{attribute 'GeneratedUsingTerminal: KL3351'}
{attribute addProperty BoxType "KL3351"}
{attribute addProperty Description ""}
{attribute addProperty Physics ""}
{attribute addProperty Id "Channel_1AT %Q*Channel_2DA3FF3C0"}
{attribute addProperty CRC "862158000"}
{attribute addProperty Size "0"}
TYPE KL3351_33637CB0 :
STRUCT
	{attribute addProperty Name "Channel_1"}
	Channel_1 : Channel_2DA3FF3C;
END_STRUCT
END_TYPE

(* stored: Version 1.2.0.0, ProductVersion 3.1.4024.11
   DUT KL3351_33637CB0: Id {960b3604-cd61-4a0b-be74-444d3aa64506} *)
